FUNCTION_BLOCK CU00xExampleCompositComponent EXTENDS TcoCore.TcoComponent
VAR_INPUT
END_VAR
VAR_OUTPUT
END_VAR
VAR
END_VAR

END_FUNCTION_BLOCK

(* stored: Version 1.1.0.1
   POU CU00xExampleCompositComponent: Id {d583945b-540e-4c57-bcdb-eea455c1874b}, SpecialFunc None *)
